DATA_BLOCK "ST10_Stopper_InterfaceDB"
VAR
  aDev : Array[1..5] of "ST_Stopper";
  Command : Array[1..5] of "UDT_Stopper_FB";
END_VAR
BEGIN
END_DATA_BLOCK
